FUNCTION_BLOCK catTest (* CAT Function Block Type *)
  (* Standard: 61499-2 *)
  (* Version 0.0, 10/2/2026, Schneider Electric, template *)
  PACKAGE Main;
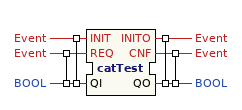
  EVENT_INPUT
    INIT WITH QI; (* Initialization Request *)
    REQ WITH QI; (* Normal Execution Request *)
  END_EVENT
  EVENT_OUTPUT
    INITO WITH QO; (* Initialization Confirm *)
    CNF WITH QO; (* Execution Confirmation *)
  END_EVENT
  VAR_INPUT
    QI : BOOL; (* Input event qualifier *)
  END_VAR
  VAR_OUTPUT
    QO : BOOL; (* Output event qualifier *)
  END_VAR
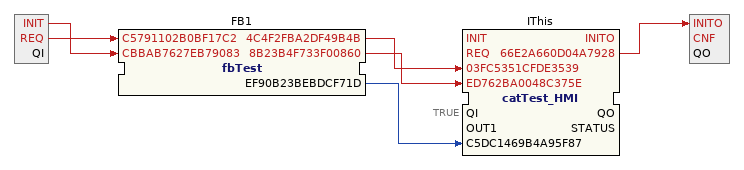
  FBS
    FB1 : fbTest;
    IThis : catTest_HMI(QI := TRUE);
  END_FBS
  EVENT_CONNECTIONS
    REQ TO FB1.C5791102B0BF17C2;
    INIT TO FB1.CBBAB7627EB79083;
    FB1.4C4F2FBA2DF49B4B TO IThis.03FC5351CFDE3539;
    FB1.8B23B4F733F00860 TO IThis.ED762BA0048C375E;
    IThis.66E2A660D04A7928 TO INITO;
  END_CONNECTIONS
  DATA_CONNECTIONS
    FB1.EF90B23BEBDCF71D TO IThis.C5DC1469B4A95F87;
  END_CONNECTIONS
END_FUNCTION_BLOCK
